// TIA Portal V18 export
DATA_BLOCK "L1_packetdata"   // DB27
{ S7_Optimized_Access := 'TRUE' }
VERSION : 0.1
// stored: AutoNumber false, DBAccessibleFromOPCUA true, DBAccessibleFromWebserver false, IsOnlyStoredInLoadMemory false, IsRetainMemResEnabled false, IsWriteProtectedInAS false, MemoryReserve 100
   VAR RETAIN
      pz : Array[1..200] of "LGasp_Type_packetdata";
   END_VAR
BEGIN
END_DATA_BLOCK
